% RSLogix 500 project Test Prog.RSS, saved by version 11.00.00.00 %
PROJECT "UNTITLED"    % processor: MicroLogix 1400 %

PROGRAM FILES
  LAD 2   2 rungs

DATA FILES
  O0 OUTPUT  6 elements
  I1 INPUT  8 elements
  S2 STATUS  66 elements
  B3 BINARY  1 elements
  T4 TIMER  1 elements
  C5 COUNTER  1 elements
  R6 CONTROL  1 elements
  N7 INTEGER  1 elements
  F8 FLOAT  1 elements

LADDER 2
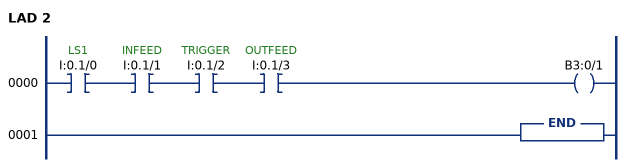
% Rung: 0 %
SOR XIC I:0.1/0 XIC I:0.1/1 XIC I:0.1/2 XIC I:0.1/3 OTE B3:0/1 EOR
%   I:0.1/0  LS1 %
%   I:0.1/1  INFEED %
%   I:0.1/2  TRIGGER %
%   I:0.1/3  OUTFEED %
% Rung: 1 %
SOR END EOR
